(* IEC 61131-3 sources: automationbase/test/Equipment, 5 files *)

(* ---- StartUpStatusAssert.st ---- *)
USING AxUnit.ResultFunctions;
USING Simatic.Ax.AutomationBase;
USING System.Strings;

NAMESPACE Simatic.Ax.AutomationBase

    /// <summary>
    /// Custom assertion function for comparing StartUpStatus enum values.
    /// Provides clear error messages showing expected vs actual values with enum names.
    /// </summary>
    /// <param name="expected">The expected StartUpStatus value</param>
    /// <param name="actual">The actual StartUpStatus value to compare</param>
    /// <param name="file">Caller file path (automatically filled by compiler)</param>
    /// <param name="line">Caller line number (automatically filled by compiler)</param>
    FUNCTION PUBLIC EqualStartUpStatus
        VAR_INPUT
            expected : StartUpStatus;
            actual : StartUpStatus;
            {CallerFilePath}
            file : WSTRING[1024];
            {CallerLineNumber}
            line : INT;
        END_VAR
        VAR_TEMP
            message : STRING[254];
        END_VAR

        // If values match, test passes
        IF expected = actual THEN
            axunit_Succeed();
        ELSE
            // Build descriptive error message with enum names
            message := 'Expected StartUpStatus to be ';
            CASE expected OF
                StartUpStatus#InternalError:
                    message := Concat(message, 'InternalError');
                StartUpStatus#NotReleased:
                    message := Concat(message, 'NotReleased');
                StartUpStatus#AutoStartingUp:
                    message := Concat(message, 'AutoStartingUp');
                StartUpStatus#AutoStartedUp:
                    message := Concat(message, 'AutoStartedUp');
            END_CASE;
            message := Concat(message, ' but was ');
            CASE actual OF
                StartUpStatus#InternalError:
                    message := Concat(message, 'InternalError');
                StartUpStatus#NotReleased:
                    message := Concat(message, 'NotReleased');
                StartUpStatus#AutoStartingUp:
                    message := Concat(message, 'AutoStartingUp');
                StartUpStatus#AutoStartedUp:
                    message := Concat(message, 'AutoStartedUp');
            END_CASE;
            // Report test failure with descriptive message
            axunit_Fail(message, file, line);
        END_IF;
    END_FUNCTION

END_NAMESPACE

(* ---- EquipmentAutoStartupTest.st ---- *)
USING Simatic.Ax.Conveyor.Mocks;
USING Simatic.Ax.Conveyor;
USING AxUnit.Assert;
USING Simatic.Ax.AutomationBase;
NAMESPACE Simatic.Ax.AutomationBase
    {TestFixture}
    CLASS EquipmentAutoStartupTest
        VAR
            startup, startupStateless : EquipmentAutoStartup;
            mockMan, mockManStateless : MockOperatingMode;
            relTrue : MockIsReleased_TRUE;
            relFalse : MockIsReleased_FALSE;
            mockEquipment, mockEquipmentStateless : MockEquiment;
        END_VAR

        {TestSetup}
        METHOD PUBLIC TestSetup
            startup := startupStateless;
            mockEquipment := mockEquipmentStateless;
            mockMan := mockManStateless;
        END_METHOD

        {Test}
        METHOD PUBLIC StartupProhibitedOfError
            mockMan.mode := OperatingModes#Automatic;
            startup.Mode := mockMan;
            startup.Release := relTrue;
            startup.equipment := mockEquipment;
            mockEquipment.MockError := TRUE;

            startup.RunCyclic();
            Equal(expected := TRUE , actual := startup.Status() = StartUpStatus#NotReleased);
        END_METHOD
        {Test}
        METHOD PUBLIC StartupProhibitedOfNoRelease
            mockMan.mode := OperatingModes#Automatic;
            startup.Mode := mockMan;
            startup.Release := relFalse;
            startup.equipment := mockEquipment;

            startup.RunCyclic();
            Equal(expected := TRUE , actual := startup.Status() = StartUpStatus#NotReleased);
        END_METHOD
        {Test}
        METHOD PUBLIC StartupProhibitedOfNoAutomatic
            mockMan.mode := OperatingModes#Commissioning;
            startup.Mode := mockMan;
            startup.Release := relTrue;
            startup.equipment := mockEquipment;

            startup.RunCyclic();
            Equal(expected := TRUE , actual := startup.Status() = StartUpStatus#NotReleased);
        END_METHOD

        {Test}
        METHOD PUBLIC Startup_InProgress_after_switch_to_automatic
            mockMan.mode := OperatingModes#Commissioning;
            startup.Mode := mockMan;
            startup.Release := relTrue;
            startup.equipment := mockEquipment;
            startup.RunCyclic();
            Equal(expected := TRUE , actual := startup.Status() = StartUpStatus#NotReleased);

            mockMan.mode := OperatingModes#Automatic;
            startup.RunCyclic();
            Equal(expected := TRUE , actual := startup.Status() = StartUpStatus#AutoStartingUp);
        END_METHOD
        {Test}
        METHOD PUBLIC When_Automatic_And_No_Release_configured_returns_AutoStartingUp
            mockMan.mode := OperatingModes#Automatic;
            startup.Mode := mockMan;
            startup.Release := NULL;
            startup.equipment := mockEquipment;
            startup.RunCyclic();
            Equal(expected := TRUE , actual := startup.Status() = StartUpStatus#AutoStartingUp);
        END_METHOD
        {Test}
        METHOD PUBLIC NotConfigured_Mode_returns_internalerror
            startup.Mode := NULL;
            startup.Release := relTrue;
            startup.equipment := mockEquipment;
            startup.RunCyclic();
            Equal(expected := TRUE , actual := startup.Status() = StartUpStatus#InternalError);
        END_METHOD
        {Test}
        METHOD PUBLIC NotConfigured_Equipment_returns_internalerror
            startup.Mode := mockMan;
            startup.Release := relTrue;
            startup.equipment := NULL;
            startup.RunCyclic();
            Equal(expected := TRUE , actual := startup.Status() = StartUpStatus#InternalError);
        END_METHOD

        {Test}
        METHOD PUBLIC Manual_Mode_returns_Manual_Status
            mockMan.mode := OperatingModes#Manual;
            startup.Mode := mockMan;
            startup.Release := relTrue;
            startup.equipment := mockEquipment;

            startup.RunCyclic();
            Equal(expected := TRUE , actual := startup.Status() = StartUpStatus#Manual);
        END_METHOD

        {Test}
        METHOD PUBLIC Manual_Mode_with_Error_returns_Manual_Status
            mockMan.mode := OperatingModes#Manual;
            startup.Mode := mockMan;
            startup.Release := relTrue;
            startup.equipment := mockEquipment;
            mockEquipment.MockError := TRUE;

            startup.RunCyclic();
            Equal(expected := TRUE , actual := startup.Status() = StartUpStatus#Manual);
        END_METHOD

        {Test}
        METHOD PUBLIC Manual_Mode_without_Release_returns_Manual_Status
            mockMan.mode := OperatingModes#Manual;
            startup.Mode := mockMan;
            startup.Release := relFalse;
            startup.equipment := mockEquipment;

            startup.RunCyclic();
            Equal(expected := TRUE , actual := startup.Status() = StartUpStatus#Manual);
        END_METHOD

        {Test}
        METHOD PUBLIC Switch_from_Manual_to_Automatic_starts_Startup
            // First set to Manual
            mockMan.mode := OperatingModes#Manual;
            startup.Mode := mockMan;
            startup.Release := relTrue;
            startup.equipment := mockEquipment;
            startup.RunCyclic();
            Equal(expected := TRUE , actual := startup.Status() = StartUpStatus#Manual);

            // Switch to Automatic
            mockMan.mode := OperatingModes#Automatic;
            startup.RunCyclic();
            Equal(expected := TRUE , actual := startup.Status() = StartUpStatus#AutoStartingUp);
        END_METHOD

        {Test}
        METHOD PUBLIC Switch_from_Automatic_to_Manual_stops_Startup
            // First set to Automatic and start startup
            mockMan.mode := OperatingModes#Automatic;
            startup.Mode := mockMan;
            startup.Release := relTrue;
            startup.equipment := mockEquipment;
            startup.RunCyclic();
            Equal(expected := TRUE , actual := startup.Status() = StartUpStatus#AutoStartingUp);

            // Switch to Manual
            mockMan.mode := OperatingModes#Manual;
            startup.RunCyclic();
            Equal(expected := TRUE , actual := startup.Status() = StartUpStatus#Manual);
        END_METHOD
    END_CLASS

END_NAMESPACE

(* ---- EquipmentBaseTest.st ---- *)
USING Simatic.Ax.Conveyor.Mocks;
USING AxUnit.Assert;
USING AutomationBase.Tests;

NAMESPACE Simatic.Ax.AutomationBase

    /// <summary>
    /// Comprehensive test suite for the EquipmentBase abstract class.
    /// Tests initialization, cyclic execution, error handling, startup status,
    /// and various configuration scenarios.
    /// </summary>
    {TestFixture}
    CLASS EquipmentBaseTest
        VAR
            // Test equipment instance and stateless backup for reset between tests
            equipment, equipmentStateless : MockEquipmentBase;
            // Mock operating mode and stateless backup
            mockMode, mockModeStateless : MockOperatingMode;
            // Mock release that always returns TRUE
            releaseTrue : MockIsReleased_TRUE;
            // Mock release that always returns FALSE
            releaseFalse : MockIsReleased_FALSE;
            // Mock auto startup and stateless backup
            mockAutoStartup, mockAutoStartupStateless : MockAutoStartup;
        END_VAR

        /// <summary>
        /// Setup method executed before each test.
        /// Resets all test instances to stateless state and clears tracking flags.
        /// </summary>
        {TestSetup}
        METHOD PUBLIC TestSetup
            // Reset to stateless instances for clean state
            equipment := equipmentStateless;
            mockMode := mockModeStateless;
            mockAutoStartup := mockAutoStartupStateless;
            // Clear all test tracking flags
            equipment.ResetTestFlags();
        END_METHOD

        // ========================================
        // Initialization Tests
        // ========================================

        /// <summary>
        /// Test: Verifies that Init() calls the abstract InitUser() method.
        /// This ensures derived classes can perform custom initialization.
        /// </summary>
        {Test}
        METHOD PUBLIC Init_Calls_InitUser
            // Arrange: Setup valid configuration
            equipment.Mode := mockMode;
            mockMode.mode := OperatingModes#Automatic;

            // Act: Initialize equipment via RunCyclic (Init is private)
            equipment.RunCyclic();

            // Assert: InitUser should have been called
            Equal(expected := TRUE, actual := equipment.InitUserCalled);
        END_METHOD

        /// <summary>
        /// Test: Verifies that initialization only happens once.
        /// Subsequent calls to RunCyclic should not trigger Init again.
        /// </summary>
        {Test}
        METHOD PUBLIC Init_Sets_IsInitialized_Flag
            // Arrange: Setup valid configuration
            equipment.Mode := mockMode;
            mockMode.mode := OperatingModes#Automatic;

            // Act: Initialize equipment
            equipment.RunCyclic();

            // Verify by calling RunCyclic - should not call Init again
            equipment.ResetTestFlags();
            equipment.RunCyclic();

            // Assert: InitUser should NOT be called again
            Equal(expected := FALSE, actual := equipment.InitUserCalled);
        END_METHOD

        /// <summary>
        /// Test: Verifies that missing Mode configuration sets ConfigError.
        /// Equipment requires a valid operating mode to function.
        /// </summary>
        {Test}
        METHOD PUBLIC Init_Without_Mode_Sets_ConfigError
            // Arrange: Set Mode to NULL (invalid configuration)
            equipment.Mode := NULL;

            // Act: Attempt to initialize via RunCyclic (Init is private)
            equipment.RunCyclic();

            // Assert: Should have error state
            Equal(expected := TRUE, actual := equipment.HasError());
        END_METHOD

        /// <summary>
        /// Test: Verifies that external auto startup is used when provided.
        /// This allows custom startup behavior to override the default.
        /// </summary>
        {Test}
        METHOD PUBLIC Init_With_ExternalAutoStartup_Uses_External
            // Arrange: Setup with external auto startup
            equipment.Mode := mockMode;
            mockMode.mode := OperatingModes#Automatic;
            mockAutoStartup.startupStatus := StartUpStatus#NotReleased;
            equipment.ExternalAutoStartup := mockAutoStartup;

            // Act: Initialize equipment via RunCyclic (Init is private)
            equipment.RunCyclic();

            // Assert: Should initialize successfully with external startup
            Equal(expected := TRUE, actual := equipment.InitUserCalled);
        END_METHOD

        /// <summary>
        /// Test: Verifies that default auto startup is used when external is NULL.
        /// This is the standard behavior for most equipment.
        /// </summary>
        {Test}
        METHOD PUBLIC Init_Without_ExternalAutoStartup_Uses_Default
            // Arrange: Setup without external auto startup
            equipment.Mode := mockMode;
            mockMode.mode := OperatingModes#Automatic;
            equipment.ExternalAutoStartup := NULL;
            equipment.ExternalRelease := releaseTrue;

            // Act: Initialize equipment via RunCyclic (Init is private)
            equipment.RunCyclic();

            // Assert: Should initialize successfully with default startup
            Equal(expected := TRUE, actual := equipment.InitUserCalled);
        END_METHOD

        // ========================================
        // RunCyclic Tests
        // ========================================

        /// <summary>
        /// Test: Verifies that RunCyclic automatically calls Init on first execution.
        /// This ensures equipment is always initialized before running user code.
        /// </summary>
        {Test}
        METHOD PUBLIC RunCyclic_Calls_Init_On_First_Call
            // Arrange: Setup valid configuration
            equipment.Mode := mockMode;
            mockMode.mode := OperatingModes#Automatic;

            // Act: Call RunCyclic without explicit Init
            equipment.RunCyclic();

            // Assert: Init should have been called automatically
            Equal(expected := TRUE, actual := equipment.InitUserCalled);
        END_METHOD

        /// <summary>
        /// Test: Verifies that RunCyclic executes the abstract RunCyclicUserCode method.
        /// This is where derived classes implement their cyclic logic.
        /// </summary>
        {Test}
        METHOD PUBLIC RunCyclic_Calls_RunCyclicUserCode
            // Arrange: Setup valid configuration
            equipment.Mode := mockMode;
            mockMode.mode := OperatingModes#Automatic;

            // Act: Execute one cycle
            equipment.RunCyclic();

            // Assert: User code should have been executed
            Equal(expected := TRUE, actual := equipment.RunCyclicUserCodeCalled);
        END_METHOD

        /// <summary>
        /// Test: Verifies that user code is not executed when ConfigError is set.
        /// This prevents equipment from running in an invalid configuration state.
        /// </summary>
        {Test}
        METHOD PUBLIC RunCyclic_Does_Not_Call_UserCode_On_ConfigError
            // Arrange: Create invalid configuration (NULL mode causes ConfigError)
            equipment.Mode := NULL;

            // Act: Attempt to run cyclic
            equipment.RunCyclic();

            // Assert: User code should NOT be executed
            Equal(expected := FALSE, actual := equipment.RunCyclicUserCodeCalled);
        END_METHOD

        /// <summary>
        /// Test: Verifies that initialization only happens once across multiple cycles.
        /// Repeated calls to RunCyclic should not re-initialize the equipment.
        /// </summary>
        {Test}
        METHOD PUBLIC RunCyclic_Multiple_Calls_Only_Init_Once
            // Arrange: Setup valid configuration
            equipment.Mode := mockMode;
            mockMode.mode := OperatingModes#Automatic;

            // Act: Execute multiple cycles
            equipment.RunCyclic();
            equipment.RunCyclic();
            equipment.RunCyclic();

            // Assert: Init should have been called exactly once
            Equal(expected := 1, actual := equipment.InitUserCallCount);
        END_METHOD

        /// <summary>
        /// Test: Verifies that user code executes on every cycle.
        /// Each call to RunCyclic should execute RunCyclicUserCode once.
        /// </summary>
        {Test}
        METHOD PUBLIC RunCyclic_Multiple_Calls_Execute_UserCode_Multiple_Times
            // Arrange: Setup valid configuration
            equipment.Mode := mockMode;
            mockMode.mode := OperatingModes#Automatic;

            // Act: Execute three cycles
            equipment.RunCyclic();
            equipment.RunCyclic();
            equipment.RunCyclic();

            // Assert: User code should have been called three times
            Equal(expected := 3, actual := equipment.RunCyclicUserCodeCallCount);
        END_METHOD

        // ========================================
        // Error Handling Tests
        // ========================================

        /// <summary>
        /// Test: Verifies that equipment has no error in initial state.
        /// Fresh equipment instances should start without errors.
        /// </summary>
        {Test}
        METHOD PUBLIC HasError_Returns_False_Initially
            // Assert: No error should be present initially
            Equal(expected := FALSE, actual := equipment.HasError());
        END_METHOD

        /// <summary>
        /// Test: Verifies that HasError returns TRUE after SetError is called.
        /// This confirms error state tracking works correctly.
        /// </summary>
        {Test}
        METHOD PUBLIC HasError_Returns_True_After_SetError
            // Arrange: Initialize equipment
            equipment.Mode := mockMode;
            mockMode.mode := OperatingModes#Automatic;
            equipment.RunCyclic();

            // Act: Set an error state
            equipment.SetError(errorState := ErrorState#OtherError);
            equipment.RunCyclic(); // Update _hasError flag

            // Assert: Error should be detected
            Equal(expected := TRUE, actual := equipment.HasError());
        END_METHOD

        /// <summary>
        /// Test: Verifies that SetError properly sets the error state.
        /// Tests with ConfigError specifically.
        /// </summary>
        {Test}
        METHOD PUBLIC SetError_Sets_Error_State
            // Arrange: Initialize equipment
            equipment.Mode := mockMode;
            mockMode.mode := OperatingModes#Automatic;
            equipment.RunCyclic();

            // Act: Set configuration error
            equipment.SetError(errorState := ErrorState#ConfigError);
            equipment.RunCyclic(); // Update _hasError flag

            // Assert: Error should be present
            Equal(expected := TRUE, actual := equipment.HasError());
        END_METHOD

        {Test}
        /// <summary>
        /// Test: Verifies that GetError returns NoError by default.
        /// Fresh equipment should have no error code set.
        /// </summary>
        METHOD PUBLIC GetError_Returns_NoError_By_Default
            VAR
                errorCode : WORD;
            END_VAR

            // Act: Get error code
            errorCode := equipment.GetError();

            // Assert: Should be NoError
            Equal(expected := ErrorState#NoError, actual := errorCode);
        END_METHOD

        /// <summary>
        /// Test: Verifies that GetError returns the correct error code after SetError.
        /// </summary>
        {Test}
        METHOD PUBLIC GetError_Returns_Set_Error_Code
            VAR
                errorCode : WORD;
            END_VAR

            // Act: Set an error and get it back
            equipment.SetError(errorState := ErrorState#OtherError);
            errorCode := equipment.GetError();

            // Assert: Should return the set error code
            Equal(expected := ErrorState#OtherError, actual := errorCode);
        END_METHOD

        /// <summary>
        /// Test: Verifies that SetError with error text stores the message.
        /// </summary>
        {Test}
        METHOD PUBLIC SetError_With_Text_Stores_Message
            VAR
                errorText : STRING[30];
            END_VAR

            // Act: Set error with text
            equipment.SetError(errorState := ErrorState#OtherError, errorText := 'Motor overload');
            errorText := equipment.GetErrorText();

            // Assert: Error text should be stored
            Equal(expected := 'Motor overload', actual := errorText);
        END_METHOD

        /// <summary>
        /// Test: Verifies that SetError without text clears the error message.
        /// </summary>
        {Test}
        METHOD PUBLIC SetError_Without_Text_Clears_Message
            VAR
                errorText : STRING[30];
            END_VAR

            // Arrange: Set error with text first
            equipment.SetError(errorState := ErrorState#OtherError, errorText := 'Initial error');

            // Act: Set new error without text
            equipment.SetError(errorState := ErrorState#ConfigError);
            errorText := equipment.GetErrorText();

            // Assert: Error text should be empty
            Equal(expected := '', actual := errorText);
        END_METHOD

        /// <summary>
        /// Test: Verifies that GetErrorText returns empty string by default.
        /// </summary>
        {Test}
        METHOD PUBLIC GetErrorText_Returns_Empty_By_Default
            VAR
                errorText : STRING[30];
            END_VAR

            // Act: Get error text without setting error
            errorText := equipment.GetErrorText();

            // Assert: Should be empty
            Equal(expected := '', actual := errorText);
        END_METHOD

        /// <summary>
        /// Test: Verifies that ResetFault clears the error state.
        /// </summary>
        {Test}
        METHOD PUBLIC ResetFault_Clears_Error_State
            // Arrange: Set an error
            equipment.SetError(errorState := ErrorState#OtherError);

            // Act: Reset fault
            equipment.ResetFault();

            // Assert: Error should be cleared
            Equal(expected := FALSE, actual := equipment.HasError());
        END_METHOD

        /// <summary>
        /// Test: Verifies that ResetFault clears the error message.
        /// </summary>
        {Test}
        METHOD PUBLIC ResetFault_Clears_Error_Message
            VAR
                errorText : STRING[30];
            END_VAR

            // Arrange: Set error with text
            equipment.SetError(errorState := ErrorState#OtherError, errorText := 'Test error');

            // Act: Reset fault
            equipment.ResetFault();
            errorText := equipment.GetErrorText();

            // Assert: Error text should be cleared
            Equal(expected := '', actual := errorText);
        END_METHOD

        /// <summary>
        /// Test: Verifies that ResetFault clears both error code and message.
        /// </summary>
        {Test}
        METHOD PUBLIC ResetFault_Clears_Both_Error_And_Message
            VAR
                errorCode : WORD;
                errorText : STRING[30];
            END_VAR

            // Arrange: Set error with text
            equipment.SetError(errorState := ErrorState#OtherError, errorText := 'Critical fault');

            // Act: Reset fault
            equipment.ResetFault();
            errorCode := equipment.GetError();
            errorText := equipment.GetErrorText();

            // Assert: Both should be cleared
            Equal(expected := ErrorState#NoError, actual := errorCode);
            Equal(expected := '', actual := errorText);
        END_METHOD

        // ========================================
        // Startup Status Tests
        // ========================================

        /// <summary>
        /// Test: Verifies that GetStartupStatus returns InternalError before initialization.
        /// Uninitialized equipment cannot provide valid startup status.
        /// </summary>
        {Test}
        METHOD PUBLIC GetStartupStatus_Returns_InternalError_Before_Init
            VAR
                status : StartUpStatus;
            END_VAR

            // Act: Get status without initialization
            status := equipment.GetStartupStatus();

            // Assert: Should return InternalError
            EqualStartUpStatus(expected := StartUpStatus#InternalError, actual := status);
        END_METHOD

        /// <summary>
        /// Test: Verifies that GetStartupStatus returns valid status after initialization.
        /// Once initialized, equipment should provide meaningful startup status.
        /// </summary>
        {Test}
        METHOD PUBLIC GetStartupStatus_Returns_Valid_After_Init
            VAR
                status : StartUpStatus;
            END_VAR
            // Arrange: Setup and initialize equipment
            equipment.Mode := mockMode;
            mockMode.mode := OperatingModes#Automatic;
            equipment.ExternalRelease := releaseTrue;

            // Act: Initialize via RunCyclic (Init is private) and get status
            equipment.RunCyclic();
            status := equipment.GetStartupStatus();

            // Assert: Should not be InternalError anymore
            Equal(expected := FALSE, actual := status = StartUpStatus#InternalError);
        END_METHOD

        /// <summary>
        /// Test: Verifies that startup status is NotReleased when release condition is false.
        /// Equipment in manual mode without release should report NotReleased status.
        /// </summary>
        {Test}
        METHOD PUBLIC GetStartupStatus_NotReleased_When_Release_Is_False
            VAR
                status : StartUpStatus;
            END_VAR
            // Arrange: Setup with manual mode and false release
            equipment.Mode := mockMode;
            mockMode.mode := OperatingModes#Manual;
            equipment.ExternalRelease := releaseFalse;

            // Act: Run cycle (initializes automatically) and get status
            equipment.RunCyclic();
            equipment.RunCyclic(); // Second cycle to ensure startup system is fully initialized
            status := equipment.GetStartupStatus();

            // Assert: Should be Manual (not NotReleased) when in Manual mode
            EqualStartUpStatus(expected := StartUpStatus#Manual, actual := status);
        END_METHOD

        // ========================================
        // Release Configuration Tests
        // ========================================

        /// <summary>
        /// Test: Verifies that external release is properly configured in default auto startup.
        /// When no external auto startup is provided, the default should use external release.
        /// </summary>
        {Test}
        METHOD PUBLIC Init_With_ExternalRelease_Configures_DefaultAutoStartup
            // Arrange: Setup with external release but no external auto startup
            equipment.Mode := mockMode;
            mockMode.mode := OperatingModes#Automatic;
            equipment.ExternalRelease := releaseTrue;
            equipment.ExternalAutoStartup := NULL;

            // Act: Initialize equipment via RunCyclic (Init is private)
            equipment.RunCyclic();

            // Assert: Should initialize successfully
            Equal(expected := TRUE, actual := equipment.InitUserCalled);
        END_METHOD

        /// <summary>
        /// Test: Verifies null-object pattern for release.
        /// When no external release is provided, equipment uses AlwaysReleased internally.
        /// </summary>
        {Test}
        METHOD PUBLIC Init_Without_ExternalRelease_Uses_AlwaysReleased
            // Arrange: Setup without external release or auto startup
            equipment.Mode := mockMode;
            mockMode.mode := OperatingModes#Automatic;
            equipment.ExternalRelease := NULL;
            equipment.ExternalAutoStartup := NULL;

            // Act: Initialize equipment via RunCyclic (Init is private)
            equipment.RunCyclic();

            // Assert: Should initialize successfully with null-object pattern
            Equal(expected := TRUE, actual := equipment.InitUserCalled);
        END_METHOD

        // ========================================
        // StartUpTime Configuration Tests
        // ========================================

        /// <summary>
        /// Test: Verifies that default startup time is 5 seconds.
        /// This is the standard startup warning time for equipment.
        /// </summary>
        {Test}
        METHOD PUBLIC StartUpTime_Default_Is_5_Seconds
            VAR
                expectedTime : TIME := T#5s;
            END_VAR

            // Assert: Default should be 5 seconds
            Equal(expected := expectedTime, actual := equipment.StartUpTime);
        END_METHOD

        /// <summary>
        /// Test: Verifies that startup time can be customized.
        /// Different equipment may require different startup warning periods.
        /// </summary>
        {Test}
        METHOD PUBLIC StartUpTime_Can_Be_Changed
            VAR
                customTime : TIME := T#10s;
            END_VAR

            // Act: Set custom startup time
            equipment.StartUpTime := customTime;

            // Assert: Should reflect the new value
            Equal(expected := customTime, actual := equipment.StartUpTime);
        END_METHOD

        // ========================================
        // Integration Tests
        // ========================================

        /// <summary>
        /// Test: Verifies complete lifecycle from initialization through multiple cycles.
        /// This integration test ensures all components work together correctly.
        /// </summary>
        {Test}
        METHOD PUBLIC Full_Lifecycle_Without_Errors
            // Arrange: Setup valid configuration
            equipment.Mode := mockMode;
            mockMode.mode := OperatingModes#Automatic;
            equipment.ExternalRelease := releaseTrue;

            // Act: Initialize via first RunCyclic
            equipment.RunCyclic();
            Equal(expected := TRUE, actual := equipment.InitUserCalled);

            // Act: Run multiple additional cycles
            equipment.RunCyclic();
            equipment.RunCyclic();

            // Assert: No errors and correct execution count
            Equal(expected := FALSE, actual := equipment.HasError());
            Equal(expected := 3, actual := equipment.RunCyclicUserCodeCallCount);
        END_METHOD

        /// <summary>
        /// Test: Verifies that error state prevents user code execution.
        /// When ConfigError is set, equipment should not execute cyclic user code.
        /// </summary>
        {Test}
        METHOD PUBLIC Error_State_Prevents_UserCode_Execution
            // Arrange: Initialize equipment normally
            equipment.Mode := mockMode;
            mockMode.mode := OperatingModes#Automatic;

            equipment.RunCyclic();
            equipment.ResetTestFlags();

            // Act: Set config error and try to run
            equipment.SetError(errorState := ErrorState#ConfigError);
            equipment.RunCyclic();

            // Assert: UserCode should not be called
            Equal(expected := FALSE, actual := equipment.RunCyclicUserCodeCalled);
        END_METHOD

        /// <summary>
        /// Test: Verifies that equipment continues to work after mode change.
        /// Switching from Manual to Automatic should not break functionality.
        /// </summary>
        {Test}
        METHOD PUBLIC Mode_Change_From_Manual_To_Automatic
            VAR
                status : StartUpStatus;
            END_VAR
            // Arrange: Initialize in manual mode
            equipment.Mode := mockMode;
            mockMode.mode := OperatingModes#Manual;
            equipment.ExternalRelease := releaseTrue;

            equipment.RunCyclic();

            // Act: Switch to automatic mode
            mockMode.mode := OperatingModes#Automatic;
            equipment.RunCyclic();

            // Assert: Should still execute user code
            Equal(expected := TRUE, actual := equipment.RunCyclicUserCodeCalled);
        END_METHOD

    END_CLASS

END_NAMESPACE

(* ---- ResetCommandIntegrationTest.st ---- *)
NAMESPACE Simatic.Ax.AutomationBase.Test

    USING Simatic.Ax.AutomationBase;
    USING Simatic.Ax.IO.Input;
    USING AxUnit.Assert;

    /// Mock equipment for testing reset functionality
    CLASS MockEquipmentForReset EXTENDS EquipmentBase
        VAR PUBLIC
            SimulateError : BOOL;
            ResetWasCalled : BOOL;
            ResetCallCount : INT;
            CustomResetValue : INT;
        END_VAR

        METHOD PROTECTED OVERRIDE InitUser
            ResetWasCalled := FALSE;
            ResetCallCount := 0;
            CustomResetValue := 0;
        END_METHOD

        METHOD PROTECTED OVERRIDE RunCyclicUserCode
            // Simulate error condition
            IF (SimulateError AND NOT THIS.HasError()) THEN
                THIS.SetError(errorState := ErrorState#OtherError,
                             errorText := 'Test error');
            END_IF;
        END_METHOD

        METHOD PROTECTED OVERRIDE ResetFaultUser : BOOL
            // Clear error simulation flag
            SimulateError := FALSE;

            // Custom test logic
            ResetWasCalled := TRUE;
            ResetCallCount := ResetCallCount + 1;
            CustomResetValue := 42; // Test value to verify custom reset

            ResetFaultUser := TRUE;
        END_METHOD
    END_CLASS

    {TestFixture}
    CLASS ResetCommandIntegrationTest
        VAR PROTECTED
            equipment1, equipment1Stateless : MockEquipmentForReset;
            equipment2, equipment2Stateless : MockEquipmentForReset;
            equipment3, equipment3Stateless : MockEquipmentForReset;
            resetManager, resetManagerStateless : ResetCommandManager;
            modeManager, modeManagerStateless : OperatingModeManager;
            binSignal, binSignalStateless : BinSignal;
        END_VAR

        {TestSetup}
        METHOD PUBLIC Setup
            // Reset to stateless instances
            equipment1 := equipment1Stateless;
            equipment2 := equipment2Stateless;
            equipment3 := equipment3Stateless;
            resetManager := resetManagerStateless;
            modeManager := modeManagerStateless;
            binSignal := binSignalStateless;

            // Connect signal to reset manager
            resetManager.ResetSignal := binSignal;

            // Configure equipment
            equipment1.Mode := modeManager;
            equipment1.ResetCommand := resetManager;

            equipment2.Mode := modeManager;
            equipment2.ResetCommand := resetManager;

            equipment3.Mode := modeManager;
            equipment3.ResetCommand := resetManager;

            // Initialize equipment
            equipment1.RunCyclic();
            equipment2.RunCyclic();
            equipment3.RunCyclic();
            resetManager.RunCyclic();
        END_METHOD

        {Test}
        METHOD PUBLIC Test_SingleEquipmentWithError_ResetsSuccessfully
            // Arrange: Equipment 1 has error
            equipment1.SimulateError := TRUE;
            equipment1.RunCyclic(); // Sets error in user code
            equipment1.RunCyclic(); // Updates _hasError flag
            resetManager.RunCyclic();
            Equal(actual := equipment1.HasError(), expected := TRUE);
            Equal(actual := resetManager.AnyErrorActive(), expected := TRUE);

            // Establish signal state and trigger reset
            binSignal.ReadCyclic(signal := FALSE, valid := TRUE);
            resetManager.RunCyclic();

            binSignal.ReadCyclic(signal := TRUE, valid := TRUE);
            resetManager.RunCyclic();

            equipment1.RunCyclic();
            equipment2.RunCyclic();
            equipment3.RunCyclic();
            resetManager.RunCyclic();

            // Assert: Error cleared and custom reset called
            Equal(actual := equipment1.HasError(), expected := FALSE);
            Equal(actual := equipment1.ResetWasCalled, expected := TRUE);
            Equal(actual := equipment1.ResetCallCount, expected := 1);
            Equal(actual := equipment1.CustomResetValue, expected := 42);
            Equal(actual := resetManager.AnyErrorActive(), expected := FALSE);
        END_METHOD

        {Test}
        METHOD PUBLIC Test_MultipleEquipmentWithErrors_AllReset
            // Arrange: All equipment have errors
            equipment1.SimulateError := TRUE;
            equipment2.SimulateError := TRUE;
            equipment3.SimulateError := TRUE;

            equipment1.RunCyclic(); // Sets error
            equipment2.RunCyclic(); // Sets error
            equipment3.RunCyclic(); // Sets error
            equipment1.RunCyclic(); // Updates _hasError flag
            equipment2.RunCyclic(); // Updates _hasError flag
            equipment3.RunCyclic(); // Updates _hasError flag
            resetManager.RunCyclic();

            Equal(actual := equipment1.HasError(), expected := TRUE);
            Equal(actual := equipment2.HasError(), expected := TRUE);
            Equal(actual := equipment3.HasError(), expected := TRUE);
            Equal(actual := resetManager.AnyErrorActive(), expected := TRUE);

            // Establish signal state and trigger reset
            binSignal.ReadCyclic(signal := FALSE, valid := TRUE);
            resetManager.RunCyclic();

            binSignal.ReadCyclic(signal := TRUE, valid := TRUE);
            resetManager.RunCyclic();

            equipment1.RunCyclic();
            equipment2.RunCyclic();
            equipment3.RunCyclic();
            resetManager.RunCyclic();

            // Assert: All errors cleared
            Equal(actual := equipment1.HasError(), expected := FALSE);
            Equal(actual := equipment2.HasError(), expected := FALSE);
            Equal(actual := equipment3.HasError(), expected := FALSE);

            Equal(actual := equipment1.ResetWasCalled, expected := TRUE);
            Equal(actual := equipment2.ResetWasCalled, expected := TRUE);
            Equal(actual := equipment3.ResetWasCalled, expected := TRUE);

            Equal(actual := resetManager.AnyErrorActive(), expected := FALSE);
        END_METHOD

        {Test}
        METHOD PUBLIC Test_MixedEquipment_OnlyErrorsReset
            // Arrange: Only equipment 1 and 3 have errors
            equipment1.SimulateError := TRUE;
            equipment3.SimulateError := TRUE;

            equipment1.RunCyclic(); // Sets error
            equipment2.RunCyclic();
            equipment3.RunCyclic(); // Sets error
            equipment1.RunCyclic(); // Updates _hasError flag
            equipment3.RunCyclic(); // Updates _hasError flag
            resetManager.RunCyclic();

            Equal(actual := resetManager.AnyErrorActive(), expected := TRUE);

            // Establish signal state and trigger reset
            binSignal.ReadCyclic(signal := FALSE, valid := TRUE);
            resetManager.RunCyclic();

            binSignal.ReadCyclic(signal := TRUE, valid := TRUE);
            resetManager.RunCyclic();

            equipment1.RunCyclic();
            equipment2.RunCyclic();
            equipment3.RunCyclic();
            resetManager.RunCyclic();

            // Assert: Only equipment with errors called reset
            Equal(actual := equipment1.ResetWasCalled, expected := TRUE);
            Equal(actual := equipment2.ResetWasCalled, expected := FALSE); // No error, no reset
            Equal(actual := equipment3.ResetWasCalled, expected := TRUE);

            Equal(actual := resetManager.AnyErrorActive(), expected := FALSE);
        END_METHOD

        {Test}
        METHOD PUBLIC Test_NoEquipmentWithErrors_NoResets
            // Arrange: No equipment have errors
            equipment1.RunCyclic();
            equipment2.RunCyclic();
            equipment3.RunCyclic();
            resetManager.RunCyclic();

            Equal(actual := equipment1.HasError(), expected := FALSE);
            Equal(actual := equipment2.HasError(), expected := FALSE);
            Equal(actual := equipment3.HasError(), expected := FALSE);
            Equal(actual := resetManager.AnyErrorActive(), expected := FALSE);

            // Establish signal state and trigger reset
            binSignal.ReadCyclic(signal := FALSE, valid := TRUE);
            resetManager.RunCyclic();

            binSignal.ReadCyclic(signal := TRUE, valid := TRUE);
            resetManager.RunCyclic();

            equipment1.RunCyclic();
            equipment2.RunCyclic();
            equipment3.RunCyclic();
            resetManager.RunCyclic();

            // Assert: No resets called
            Equal(actual := equipment1.ResetWasCalled, expected := FALSE);
            Equal(actual := equipment2.ResetWasCalled, expected := FALSE);
            Equal(actual := equipment3.ResetWasCalled, expected := FALSE);

            Equal(actual := resetManager.AnyErrorActive(), expected := FALSE);
        END_METHOD

        {Test}
        METHOD PUBLIC Test_ResetCommand_ClearsAutomatically
            // Arrange: Equipment 1 has error
            equipment1.SimulateError := TRUE;
            equipment1.RunCyclic();
            resetManager.RunCyclic();

            // Establish signal state and trigger reset
            binSignal.ReadCyclic(signal := FALSE, valid := TRUE);
            resetManager.RunCyclic();

            binSignal.ReadCyclic(signal := TRUE, valid := TRUE);
            resetManager.RunCyclic();
            Equal(actual := resetManager.IsResetActive(), expected := TRUE);

            // Equipment resets
            binSignal.ReadCyclic(signal := FALSE, valid := TRUE);
            equipment1.RunCyclic();
            equipment2.RunCyclic();
            equipment3.RunCyclic();
            resetManager.RunCyclic();

            // Assert: Reset command cleared automatically
            Equal(actual := resetManager.IsResetActive(), expected := FALSE);
            Equal(actual := equipment1.HasError(), expected := FALSE);
        END_METHOD

        {Test}
        METHOD PUBLIC Test_MultipleResetCycles_WorkCorrectly
            // First reset cycle - establish signal state
            binSignal.ReadCyclic(signal := FALSE, valid := TRUE);
            resetManager.RunCyclic();

            equipment1.SimulateError := TRUE;
            equipment1.RunCyclic();
            resetManager.RunCyclic();

            binSignal.ReadCyclic(signal := TRUE, valid := TRUE);
            resetManager.RunCyclic();
            equipment1.RunCyclic();
            equipment2.RunCyclic();
            equipment3.RunCyclic();
            resetManager.RunCyclic();

            Equal(actual := equipment1.HasError(), expected := FALSE);
            Equal(actual := equipment1.ResetCallCount, expected := 1);

            // Second reset cycle
            binSignal.ReadCyclic(signal := FALSE, valid := TRUE);
            resetManager.RunCyclic();

            equipment1.SimulateError := TRUE;
            equipment2.SimulateError := TRUE;
            equipment1.RunCyclic();
            equipment2.RunCyclic();
            equipment3.RunCyclic();
            resetManager.RunCyclic();

            binSignal.ReadCyclic(signal := TRUE, valid := TRUE);
            resetManager.RunCyclic();
            equipment1.RunCyclic();
            equipment2.RunCyclic();
            equipment3.RunCyclic();
            resetManager.RunCyclic();

            // Assert: Both equipment reset
            Equal(actual := equipment1.HasError(), expected := FALSE);
            Equal(actual := equipment2.HasError(), expected := FALSE);
            Equal(actual := equipment1.ResetCallCount, expected := 2); // Reset twice
            Equal(actual := equipment2.ResetCallCount, expected := 1); // Reset once
        END_METHOD

        {Test}
        METHOD PUBLIC Test_EquipmentWithoutResetCommand_NotAffected
            // Arrange: Disconnect equipment3 from reset manager
            equipment3.ResetCommand := NULL;
            equipment3.SimulateError := TRUE;
            equipment3.RunCyclic();
            resetManager.RunCyclic();

            equipment1.SimulateError := TRUE;
            equipment1.RunCyclic();
            resetManager.RunCyclic();

            // Establish signal state and trigger reset
            binSignal.ReadCyclic(signal := FALSE, valid := TRUE);
            resetManager.RunCyclic();

            binSignal.ReadCyclic(signal := TRUE, valid := TRUE);
            resetManager.RunCyclic();
            equipment1.RunCyclic();
            equipment2.RunCyclic();
            equipment3.RunCyclic();
            resetManager.RunCyclic();

            // Assert: Only equipment1 reset, equipment3 still has error
            Equal(actual := equipment1.HasError(), expected := FALSE);
            Equal(actual := equipment3.HasError(), expected := TRUE); // Still has error
            Equal(actual := equipment1.ResetWasCalled, expected := TRUE);
            Equal(actual := equipment3.ResetWasCalled, expected := FALSE);
        END_METHOD

        {Test}
        METHOD PUBLIC Test_ManualResetFault_WorksIndependently
            // Arrange: Equipment has error
            equipment1.SimulateError := TRUE;
            equipment1.RunCyclic(); // Sets error
            equipment1.RunCyclic(); // Updates _hasError flag
            resetManager.RunCyclic();
            Equal(actual := equipment1.HasError(), expected := TRUE);

            // Act: Manual reset (not via ResetCommand)
            equipment1.ResetFault();

            // Assert: Error cleared and custom reset called
            Equal(actual := equipment1.HasError(), expected := FALSE);
            Equal(actual := equipment1.ResetWasCalled, expected := TRUE);
            Equal(actual := equipment1.CustomResetValue, expected := 42);
        END_METHOD

        {Test}
        METHOD PUBLIC Test_ErrorFlag_TracksCorrectly
            // Arrange: Create errors
            equipment1.SimulateError := TRUE;
            equipment2.SimulateError := TRUE;

            equipment1.RunCyclic(); // Sets error
            equipment2.RunCyclic(); // Sets error
            equipment3.RunCyclic();
            equipment1.RunCyclic(); // Updates _hasError flag
            equipment2.RunCyclic(); // Updates _hasError flag
            resetManager.RunCyclic();

            // Assert: Error flag should be active
            Equal(actual := resetManager.AnyErrorActive(), expected := TRUE);

            // Establish signal state and trigger reset
            binSignal.ReadCyclic(signal := FALSE, valid := TRUE);
            resetManager.RunCyclic();

            binSignal.ReadCyclic(signal := TRUE, valid := TRUE);
            resetManager.RunCyclic();
            equipment1.RunCyclic();
            binSignal.ReadCyclic(signal := FALSE, valid := TRUE);
            resetManager.RunCyclic();
            equipment2.SimulateError := TRUE; // Keep equipment2 error
            equipment2.RunCyclic();
            equipment3.RunCyclic();
            resetManager.RunCyclic();

            // Assert: Error flag still active because equipment2 still has error
            Equal(actual := resetManager.AnyErrorActive(), expected := TRUE);
        END_METHOD
    END_CLASS

END_NAMESPACE

(* ---- ResetCommandManagerTest.st ---- *)
NAMESPACE Simatic.Ax.AutomationBase.Test

    USING Simatic.Ax.AutomationBase;
    USING Simatic.Ax.IO.Input;
    USING AxUnit.Assert;

    {TestFixture}
    CLASS ResetCommandManagerTest
        VAR PROTECTED
            resetManager, resetManagerStateless : ResetCommandManager;
            binSignal, binSignalStateless : BinSignal;
        END_VAR

        {TestSetup}
        METHOD PUBLIC TestSetup
            // Reset to stateless instances for clean state
            resetManager := resetManagerStateless;
            binSignal := binSignalStateless;

            // Connect signal to reset manager
            resetManager.ResetSignal := binSignal;

            // Establish initial signal state (LOW)
            binSignal.ReadCyclic(signal := FALSE, valid := TRUE);
            resetManager.RunCyclic();
        END_METHOD

        {Test}
        METHOD PUBLIC Test_InitialState_NoErrorsActive
            // Assert: Initial state should have no errors
            Equal(actual := resetManager.AnyErrorActive(), expected := FALSE);
            Equal(actual := resetManager.AnyErrorActive(), expected := FALSE);
            Equal(actual := resetManager.IsResetActive(), expected := FALSE);
        END_METHOD

        {Test}
        METHOD PUBLIC Test_ReportError_SetsErrorActive
            // Act: Report an error and complete cycle
            resetManager.ReportError();
            resetManager.RunCyclic();

            // Assert: Error should be active
            Equal(actual := resetManager.AnyErrorActive(), expected := TRUE);
            Equal(actual := resetManager.AnyErrorActive(), expected := TRUE);
        END_METHOD

        {Test}
        METHOD PUBLIC Test_MultipleReportError_SetsErrorActive
            // Act: Report multiple errors and complete cycle
            resetManager.ReportError();
            resetManager.ReportError();
            resetManager.ReportError();
            resetManager.RunCyclic();

            // Assert: Error should be active
            Equal(actual := resetManager.AnyErrorActive(), expected := TRUE);
        END_METHOD

        {Test}
        METHOD PUBLIC Test_ResetSignal_ClearsErrorFlag
            // Arrange: Report an error and complete cycle
            resetManager.ReportError();
            resetManager.RunCyclic();
            Equal(actual := resetManager.AnyErrorActive(), expected := TRUE);

            // Establish signal state and trigger reset
            binSignal.ReadCyclic(signal := FALSE, valid := TRUE);
            resetManager.RunCyclic();

            binSignal.ReadCyclic(signal := TRUE, valid := TRUE);
            resetManager.RunCyclic();

            // Acknowledge reset and run cycle
            binSignal.ReadCyclic(signal := FALSE, valid := TRUE);
            resetManager.RunCyclic();

            // Assert: Reset should be cleared
            Equal(actual := resetManager.IsResetActive(), expected := FALSE);
        END_METHOD

        {Test}
        METHOD PUBLIC Test_ResetSignal_ActivatesResetCommand
            // Arrange: Establish initial signal state
            binSignal.ReadCyclic(signal := FALSE, valid := TRUE);
            resetManager.RunCyclic();

            // Act: Trigger reset via signal (rising edge)
            binSignal.ReadCyclic(signal := TRUE, valid := TRUE);
            resetManager.RunCyclic();

            // Assert: Reset command should be active
            Equal(actual := resetManager.ResetFaultRequest(), expected := TRUE);
            Equal(actual := resetManager.IsResetActive(), expected := TRUE);
        END_METHOD

        {Test}
        METHOD PUBLIC Test_ResetCommand_ClearsWhenNoErrors
            // Arrange: Establish initial signal state, then trigger reset with no errors
            binSignal.ReadCyclic(signal := FALSE, valid := TRUE);
            resetManager.RunCyclic();

            binSignal.ReadCyclic(signal := TRUE, valid := TRUE);
            resetManager.RunCyclic();
            Equal(actual := resetManager.IsResetActive(), expected := TRUE);

            // Act: Run another cycle with no errors (no acknowledgments needed)
            binSignal.ReadCyclic(signal := FALSE, valid := TRUE);
            resetManager.RunCyclic();

            // Assert: Reset command should clear (0 errors at reset, 0 acknowledgments = cleared)
            Equal(actual := resetManager.IsResetActive(), expected := FALSE);
            Equal(actual := resetManager.ResetFaultRequest(), expected := FALSE);
        END_METHOD

        {Test}
        METHOD PUBLIC Test_ResetCommand_ActiveForOneCycleOnly
            // Arrange: Establish signal state, report error, complete cycle, then trigger reset
            binSignal.ReadCyclic(signal := FALSE, valid := TRUE);
            resetManager.RunCyclic();

            resetManager.ReportError();
            resetManager.RunCyclic();

            binSignal.ReadCyclic(signal := TRUE, valid := TRUE);
            resetManager.RunCyclic();
            Equal(actual := resetManager.IsResetActive(), expected := TRUE);

            // Act: Run cyclic - reset should be cleared after one cycle
            resetManager.ReportError();
            binSignal.ReadCyclic(signal := FALSE, valid := TRUE);
            resetManager.RunCyclic();

            // Assert: Reset command cleared after one cycle, but error still active
            Equal(actual := resetManager.IsResetActive(), expected := FALSE);
            Equal(actual := resetManager.ResetFaultRequest(), expected := FALSE);
            Equal(actual := resetManager.AnyErrorActive(), expected := TRUE);
        END_METHOD

        {Test}
        METHOD PUBLIC Test_ResetSignal_ClearsErrorFlagAndResetCommand
            // Arrange: Report error and complete cycle
            resetManager.ReportError();
            resetManager.RunCyclic();
            Equal(actual := resetManager.AnyErrorActive(), expected := TRUE);

            // Establish signal state and trigger reset
            binSignal.ReadCyclic(signal := FALSE, valid := TRUE);
            resetManager.RunCyclic();

            binSignal.ReadCyclic(signal := TRUE, valid := TRUE);
            resetManager.RunCyclic();
            Equal(actual := resetManager.IsResetActive(), expected := TRUE);

            // Run cyclic again
            binSignal.ReadCyclic(signal := FALSE, valid := TRUE);
            resetManager.RunCyclic();

            // Assert: Reset and error flag should be cleared
            Equal(actual := resetManager.IsResetActive(), expected := FALSE);
            Equal(actual := resetManager.AnyErrorActive(), expected := FALSE);
        END_METHOD

        {Test}
        METHOD PUBLIC Test_EdgeDetection_OnlyTriggersOnRisingEdge
            VAR_TEMP
                firstCheck : BOOL;
                secondCheck : BOOL;
            END_VAR

            // Arrange: Establish initial signal state
            binSignal.ReadCyclic(signal := FALSE, valid := TRUE);
            resetManager.RunCyclic();

            // Act: Trigger reset (rising edge)
            binSignal.ReadCyclic(signal := TRUE, valid := TRUE);
            resetManager.RunCyclic();
            firstCheck := resetManager.IsResetActive();

            // Hold signal high (no rising edge)
            binSignal.ReadCyclic(signal := TRUE, valid := TRUE);
            resetManager.RunCyclic();

            // Clear reset by having no errors
            binSignal.ReadCyclic(signal := TRUE, valid := TRUE);
            resetManager.RunCyclic();
            secondCheck := resetManager.IsResetActive();

            // Assert: First trigger activates, second doesn't re-trigger
            Equal(actual := firstCheck, expected := TRUE);
            Equal(actual := secondCheck, expected := FALSE);
        END_METHOD
    END_CLASS

END_NAMESPACE
